Staubli VAL3: fileClose.pgx

program fileClose()
  local num l_nNum
begin
  for l_nNum=0 to 9
    $fileClose(l_nNum)
  endFor
  $fileClose(0)
  $fileClose(1)
  $fileClose(2)
  $fileClose(3)
  $fileClose(4)
  $fileClose(5)
  $fileClose(6)
  $fileClose(7)
  $fileClose(8)
  $fileClose(9)




end
